// TwinCAT 3 PLC project Oefening5
// ProgramVersion: 3.1.4023.0
// libraries:
//   Tc2_Standard, * (Beckhoff Automation GmbH)
//   Tc2_System, * (Beckhoff Automation GmbH)
//   Tc2_Utilities, * (Beckhoff Automation GmbH)
//   Tc3_Module, * (Beckhoff Automation GmbH)
// project tree:
//   gelijkvloers/ Gelijkvloers.TcPOU, Moving_Average.TcPOU, VISU_GVL.TcVIS
//   / GlobalTextList.TcGTLO, MAIN.TcPOU, PlcTask.TcTTO, Visualization Manager.TcVMO (not stored)
//   woning/ HOME.TcPOU, VISU_HOME.TcVIS
// (motion and I/O tree: see PLC project oefening1)
// real-time tasks:
//   TASK PlcTask: cycle T#10ms, priority 20, ADS port 350
//   TASK PlcTask1: cycle T#10ms, priority 21, ADS port 351
//   TASK PlcTask2: cycle T#10ms, priority 22, ADS port 352
//   TASK PlcTask3: cycle T#10ms, priority 23, ADS port 353
//   TASK PlcTask4: cycle T#10ms, priority 24, ADS port 354
//   TASK PlcTask5: cycle T#10ms, priority 25, ADS port 355

CONFIGURATION Oefening5
    RESOURCE PLC ON TwinCAT3
        TASK PlcTask(INTERVAL := T#10ms, PRIORITY := 25);
        PROGRAM MAIN WITH PlcTask : MAIN;
    END_RESOURCE
END_CONFIGURATION

// ---- MAIN.TcPOU
PROGRAM MAIN
VAR
END_VAR

Gelijkvloers();
Home();

END_PROGRAM

// ---- gelijkvloers/Gelijkvloers.TcPOU
PROGRAM Gelijkvloers
VAR
	TEMP_Inkom : INT;
	TEMP_Living : INT;
	TEMP_Eetruimte : INT;
	TEMP_Keuken : INT;
	TEMP_Badkamer_1 : INT;
	TEMP_Berging : INT;
	
	houseUPDATE : ARRAY [1..2, 1..6] OF INT;
	SW_Array : ARRAY [1..12] OF BOOL;
	TEMP_Keuken_Array : ARRAY [1..20] OF INT;
	
	i: INT;
	j: INT;
	
	TEMP_Buiten : INT;
	
	TON : TON;
	TOF: TOF;
	
	TON_T : TON;
	TOF_T: TOF;
	
	R_TRIG : R_TRIG;
	R_TRIG_VAR : BOOL;
END_VAR

VAR_INPUT
	SW_Inkom : BOOL;
	SW_Living : BOOL;
	SW_Eetruimte : BOOL;
	SW_Keuken : BOOL;
	SW_Badkamer_1 : BOOL;
	SW_Berging : BOOL;
	
	SW_TEMP : BOOL;
	
	SW_V_Keuken : BOOL;
	SW_V_Berging : BOOL;
	SW_V_Badkamer_1 : BOOL;
END_VAR

SW_Array[1] := SW_Inkom;
SW_Array[2] := SW_Living;
SW_Array[3] := SW_Eetruimte;
SW_Array[4] := SW_Keuken;
SW_Array[5] := SW_Berging;
SW_Array[6] := SW_Badkamer_1;

SW_Array[10] := SW_V_Keuken;
SW_Array[11] := SW_V_Berging;
SW_Array[12] := SW_V_Badkamer_1;

FOR i:=1 TO 12 BY 1 DO
	houseUpdate[1, i] := BOOL_TO_INT(SW_Array[i]);
END_FOR;

TEMP_Eetruimte := TEMP_Buiten;		
TEMP_Inkom := TEMP_Buiten;		
TEMP_Living := TEMP_Buiten;		

TOF(IN:= TON.Q, PT:= T#0MS);
TON(IN:= NOT(TOF.Q), PT:= T#3S);

IF SW_V_Keuken AND (TEMP_Keuken < 40) THEN
	TEMP_Keuken := TEMP_Keuken + BOOL_TO_INT(TOF.Q);
ELSIF (TEMP_Keuken > TEMP_BUITEN) THEN
	TEMP_Keuken := TEMP_Keuken - BOOL_TO_INT(TOF.Q);
END_IF

// Nu gaan we over naar Danny in de studio. 
TOF_T(IN:= TON_T.Q, PT:= T#0MS);
TON_T(IN:= NOT(TOF_T.Q), PT:= T#10S);

IF TOF_T.Q THEN
	FOR j:=1 TO 19 BY 1 DO
		TEMP_Keuken_Array[j] := TEMP_Keuken_Array[j+1];
	END_FOR;
	TEMP_Keuken_Array[20] := TEMP_Keuken;
END_IF

END_PROGRAM

// ---- woning/HOME.TcPOU
PROGRAM HOME
VAR
	DATA : ARRAY[1..2, 1..20] OF STRING;
	FB_LocalSystemTime : FB_LocalSystemTime;
	Moving_Average : Moving_Average;
	
	TOF : TOF;
	TON : TON;
	i : INT;
END_VAR

FB_LocalSystemTime(bEnable:= TRUE);

Moving_Average(DATA:= Gelijkvloers.TEMP_Keuken_Array);

TOF(IN:= TON.Q, PT:= T#0MS);
TON(IN:= NOT(TOF.Q), PT:= T#10S);

IF TOF.Q THEN
	FOR i:=1 TO 19 BY 1 DO
		DATA[1, i] := DATA[1, (i+1)];
		DATA[2, i] := DATA[2, (i+1)];
	END_FOR;
	DATA[1, 20] := LREAL_TO_STRING(Moving_Average.Moving_Average);
	DATA[2, 20] := SYSTEMTIME_TO_STRING(FB_LocalSystemTime.systemTime);
END_IF

END_PROGRAM

// ---- gelijkvloers/Moving_Average.TcPOU
FUNCTION_BLOCK Moving_Average

VAR_INPUT
	DATA : ARRAY[1..20] OF INT;
END_VAR

VAR_OUTPUT
	Moving_Average : LREAL;
END_VAR
VAR
	Temp_Var : LREAL;
	i: INT;
END_VAR

FOR i:=10 TO 20 BY 1 DO
	Temp_Var := (Temp_Var + DATA[i]);
END_FOR;

i := 0;
Moving_Average := Temp_Var / 10;
Temp_Var := 0;

END_FUNCTION_BLOCK

// ---- gelijkvloers/VISU_GVL.TcVIS
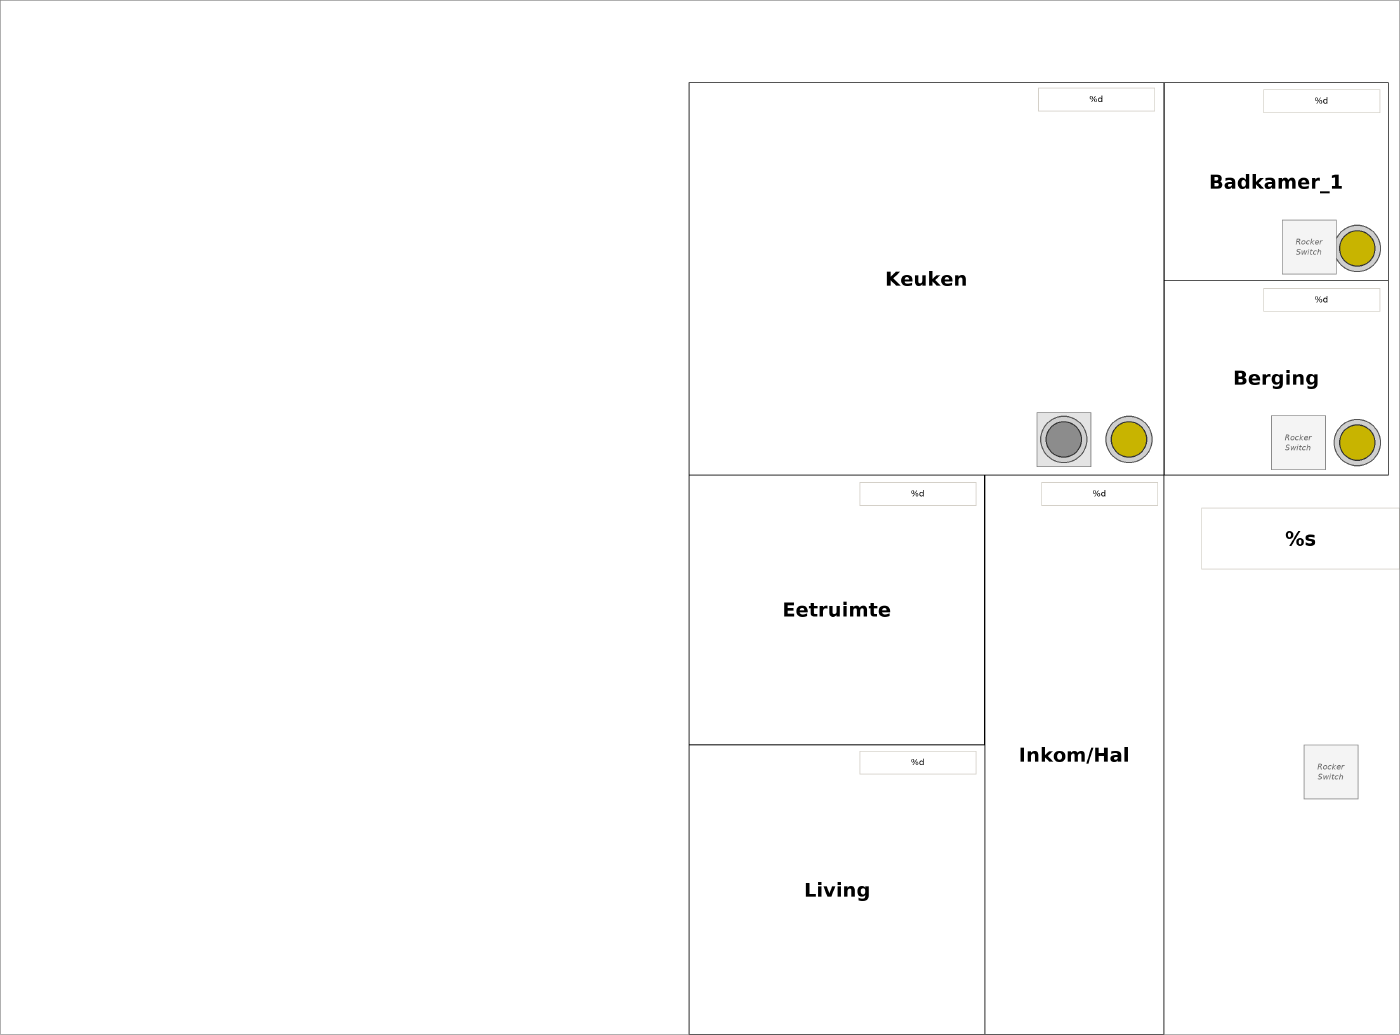
VISUALIZATION VISU_GVL  // 1803x1333
    Rectangle (887,959 383x374), "Living", colour toggle: Gelijkvloers.SW_Living
        OnMouseClick: toggle Gelijkvloers.SW_Living
    Rectangle (1268,611 231x722), "Inkom/Hal", colour toggle: Gelijkvloers.SW_Inkom
        OnMouseClick: toggle Gelijkvloers.SW_Inkom
    Rectangle (887,611 381x348), "Eetruimte", colour toggle: Gelijkvloers.SW_Eetruimte
        OnMouseClick: toggle Gelijkvloers.SW_Eetruimte
    Rectangle (887,106 612x506), "Keuken", colour toggle: Gelijkvloers.SW_Keuken
        OnMouseClick: toggle Gelijkvloers.SW_Keuken
    Rectangle (1499,106 289x256), "Badkamer_1", colour toggle: Gelijkvloers.SW_Badkamer_1
        OnMouseClick: toggle Gelijkvloers.SW_Badkamer_1
    Rectangle (1499,361 289x251), "Berging", colour toggle: Gelijkvloers.SW_Berging
        OnMouseClick: toggle Gelijkvloers.SW_Berging
    Textfield (1107,967 150x30), "%d", text variable: Gelijkvloers.TEMP_Living, invisible if: NOT Gelijkvloers.SW_TEMP
    Textfield (1107,621 150x30), "%d", text variable: Gelijkvloers.SW_Eetruimte, invisible if: NOT Gelijkvloers.SW_TEMP
    Textfield (1341,621 150x30), "%d", text variable: Gelijkvloers.TEMP_Inkom, invisible if: NOT Gelijkvloers.SW_TEMP
    Textfield (1337,113 150x30), "%d", text variable: Gelijkvloers.TEMP_Keuken, invisible if: NOT Gelijkvloers.SW_TEMP
    Textfield (1627,115 150x30), "%d", text variable: Gelijkvloers.TEMP_Badkamer_1, invisible if: NOT Gelijkvloers.SW_TEMP
    Textfield (1627,371 150x30), "%d", text variable: Gelijkvloers.TEMP_Berging, invisible if: NOT Gelijkvloers.SW_TEMP
    RockerSwitch (1679,959 70x70), variable: Gelijkvloers.SW_TEMP, behaviour: TOGGLE, style: Switch-RockerSwitch-Gray
    Lamp1 (1419,531 70x70), variable: Gelijkvloers.SW_V_Keuken, style: Lamp-Lamp1-Yellow
    Lamp1 (1713,535 70x70), variable: Gelijkvloers.SW_V_Berging, style: Lamp-Lamp1-Yellow
    Lamp1 (1713,285 70x70), variable: Gelijkvloers.SW_V_Badkamer_1, style: Lamp-Lamp1-Yellow
    RockerSwitch (1637,535 70x70), variable: Gelijkvloers.SW_V_Berging, behaviour: TOGGLE, style: Switch-RockerSwitch-Gray
    RockerSwitch (1651,283 70x70), variable: Gelijkvloers.SW_V_Badkamer_1, behaviour: TOGGLE, style: Switch-RockerSwitch-Gray
    Textfield (1547,654 256x79), "%s", text variable: Gelijkvloers.TEMP_Buiten
        OnMouseClick: write Gelijkvloers.TEMP_Buiten via Edit
    PushSwitch (1335,531 70x70), variable: Gelijkvloers.SW_V_Keuken, behaviour: TOGGLE, style: Switch-PushSwitch-Gray
END_VISUALIZATION

// ---- GlobalTextList.TcGTLO
TEXTLIST GlobalTextList
  364 = '%d'
  514 = '%s'
  273 = 'Badkamer_1'
  10 = 'Berging'
  359 = 'Eetruimte'
  146 = 'Inkom/Hal'
  347 = 'Keuken'
  708 = 'LICHT'
  120 = 'Living'
  45 = 'TEMP VAN DE KEUKEN JONGEUH'
  42 = 'VERWARMING'
END_TEXTLIST

// ---- woning/VISU_HOME.TcVIS
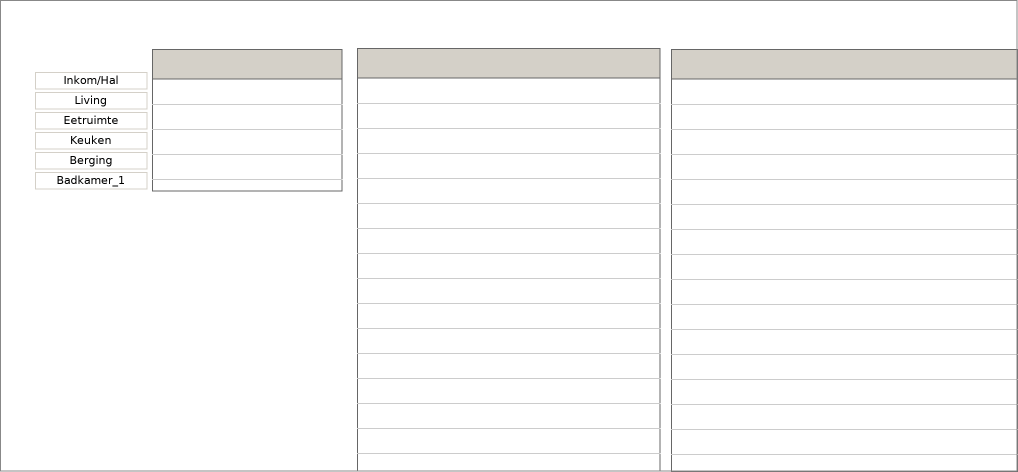
VISUALIZATION VISU_HOME  // 1018x472
    Table (152,49 190x142), data array: Gelijkvloers.houseUPDATE
        p3854506369: Gelijkvloers.houseUPDATE[1,INDEX]
        p1892666644: Gelijkvloers.houseUPDATE[2,INDEX]
    Textfield (35,72 112x17), "Inkom/Hal"
    Textfield (35,92 112x17), "Living"
    Textfield (35,112 112x17), "Eetruimte"
    Textfield (35,132 112x17), "Keuken"
    Textfield (35,152 112x17), "Berging"
    Textfield (35,172 112x17), "Badkamer_1"
    Table (357,48 303x423), data array: Gelijkvloers.TEMP_Keuken_Array
        p3854506369: Gelijkvloers.TEMP_Keuken_Array[INDEX]
        p2232123230: TEMP VAN DE KEUKEN JONGEUH
    Table (671,49 347x423), data array: HOME.DATA
        p3854506369: HOME.DATA[1,INDEX]
        p1892666644: HOME.DATA[2,INDEX]
END_VISUALIZATION
